INTERFACE BoolBindable EXTENDS BoolValue

METHOD Bind
VAR_INPUT
	boolean : REFERENCE TO BOOL;
END_VAR
END_METHOD

{attribute 'monitoring' := 'call'}
PROPERTY IsBound : BOOL
GET
END_GET
END_PROPERTY

{attribute 'monitoring' := 'call'}
PROPERTY Value : BOOL
GET
END_GET
END_PROPERTY

END_INTERFACE

(* stored: Version 1.1.0.1
   Itf BoolBindable: Id {8f04499d-19eb-4dd2-b8af-875c3c8c103f}
   Method Bind: Id {459d7cac-5a1f-4699-9462-ccea2c760ef6}
   Property IsBound: Id {bf207122-e156-4541-9506-c25dc82fbd26}
   Get Get: Id {9887206b-7c43-4055-99d6-088a465da390}
   Property Value: Id {6feaffc9-3a14-40e4-9edd-d6a719a7d44f}
   Get Get: Id {76862903-a861-4f7e-b2d3-24a8e8d88b0a} *)
